FUNCTION_BLOCK IX_Emulated (* Composite FB wrapping other FBs *)
  (* Standard: 61499-2 *)
  (* Version 1.0, 2021-08-05, dorofeev *)
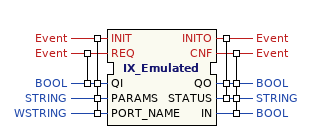
  EVENT_INPUT
    INIT WITH PARAMS, QI, PORT_NAME; (* Initialization Request *)
    REQ WITH QI; (* Normal Execution Request *)
  END_EVENT
  EVENT_OUTPUT
    INITO WITH QO, STATUS; (* Initialization Confirm *)
    CNF WITH QO, IN, STATUS; (* Execution Confirmation *)
  END_EVENT
  VAR_INPUT
    QI : BOOL; (* Input event qualifier *)
    PARAMS : STRING;
    PORT_NAME : WSTRING;
  END_VAR
  VAR_OUTPUT
    QO : BOOL; (* Output event qualifier *)
    STATUS : STRING;
    IN : BOOL;
  END_VAR
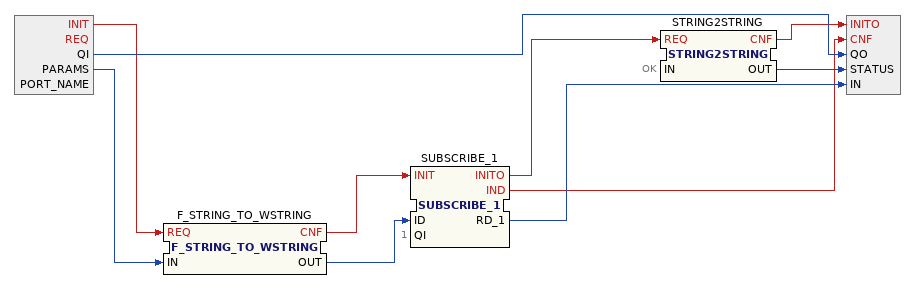
  FBS
    STRING2STRING : STRING2STRING(IN := OK);
    SUBSCRIBE_1 : SUBSCRIBE_1(QI := 1);
    F_STRING_TO_WSTRING : F_STRING_TO_WSTRING;
  END_FBS
  EVENT_CONNECTIONS
    STRING2STRING.CNF TO INITO;
    SUBSCRIBE_1.INITO TO STRING2STRING.REQ;
    SUBSCRIBE_1.IND TO CNF;
    F_STRING_TO_WSTRING.CNF TO SUBSCRIBE_1.INIT;
    INIT TO F_STRING_TO_WSTRING.REQ;
  END_CONNECTIONS
  DATA_CONNECTIONS
    STRING2STRING.OUT TO STATUS;
    SUBSCRIBE_1.RD_1 TO IN;
    QI TO QO;
    PARAMS TO F_STRING_TO_WSTRING.IN;
    F_STRING_TO_WSTRING.OUT TO SUBSCRIBE_1.ID;
  END_CONNECTIONS
END_FUNCTION_BLOCK
